(* IEC 61131-3 sources: Industry-PLC-LLM/data/PLCBEAD_repo/PLCBEAD_PLCEmbed-main/PLC-BEAD/Source/GEB/Network_TN_SC_XY2_ERROR, 1 file *)

(* ---- TN_SC_XY2_ERROR.ST ---- *)
FUNCTION TN_SC_XY2_ERROR:BOOL

	VAR_INPUT
		X1 :	INT;
		Y1 :	INT;
		X2 :	INT;
		Y2 :	INT;
	END_VAR

	TN_SC_XY2_ERROR := Y1 < 0 OR X1 < 0 OR Y2 < 0 OR X2 < 0 OR Y1 > 23 OR X1 > 79 OR Y2 > 23 OR X2 > 79;

END_FUNCTION

PROGRAM program0
	VAR
		X1 :	INT;
		Y1 :	INT;
		X2 :	INT;
		Y2 :	INT;
		CEIL5_OUT : BOOL;
	END_VAR

  	CEIL5_OUT := TN_SC_XY2_ERROR(X1, Y1, X2, Y2);
END_PROGRAM
